TYPE ST_InfoDataFB :
STRUCT
	usiMapState: USINT;
	uiMapDiag: USINT;
	usiDummy: USINT;
END_STRUCT
END_TYPE

(* stored: Version 1.1.0.1
   DUT ST_InfoDataFB: Id {9e148d4a-83e1-48a6-80d5-7617ffa625c2} *)
